// TIA Portal V20 export
FUNCTION_BLOCK "FB_Electrical_Current_Test"   // FB6, LAD
{ S7_Optimized_Access := 'TRUE' }
// stored: MemoryReserve 100, SetENOAutomatically false
   VAR_INPUT
      Star_Functional_Test : Bool;
      Reset_Functional_Test : Bool;
      Electrical_Current_Read_UInt : UInt;
      In_Test_Parameters : "IO_Device_Test_Parameters";
   END_VAR
   VAR_OUTPUT
      Electrical_Current_Test_Approved : Bool;
   END_VAR
   VAR
      Timer_Delay_Read_Current { S7_SetPoint := 'True'} : TON_TIME;
      Timer_Delay_Reset { S7_SetPoint := 'True'} : TON_TIME;
   END_VAR
BEGIN

REGION Network 1
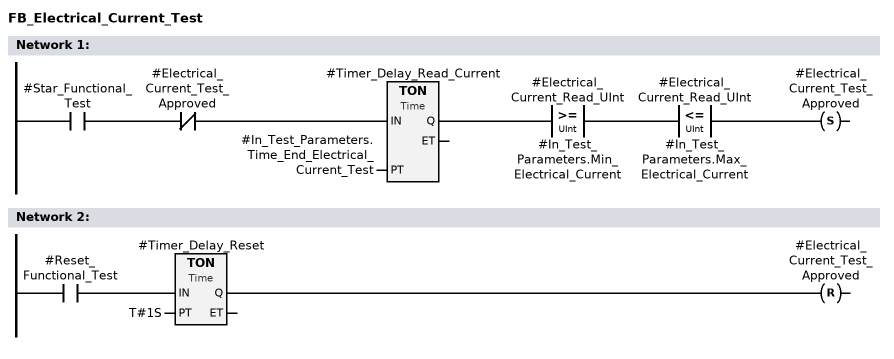
   RUNG wire#powerrail
      Contact( #Star_Functional_Test )
      I_Contact( #Electrical_Current_Test_Approved )
      { S7_Templates := "time_type := Time" } #Timer_Delay_Read_Current.TON(pt := #In_Test_Parameters.Time_End_Electrical_Current_Test, et =>)
      { S7_Templates := "SrcType := UInt" } GE_Contact(in1 := #Electrical_Current_Read_UInt, in2 := #In_Test_Parameters.Min_Electrical_Current)
      { S7_Templates := "SrcType := UInt" } LE_Contact(in1 := #Electrical_Current_Read_UInt, in2 := #In_Test_Parameters.Max_Electrical_Current)
      S_Coil( #Electrical_Current_Test_Approved )
   END_RUNG
   // the same network as SCL:
   #Timer_Delay_Read_Current(IN := #Star_Functional_Test AND NOT #Electrical_Current_Test_Approved,   // TON
                           PT := #In_Test_Parameters.Time_End_Electrical_Current_Test);
   IF #Timer_Delay_Read_Current.Q AND (#Electrical_Current_Read_UInt >= #In_Test_Parameters.Min_Electrical_Current) AND (#Electrical_Current_Read_UInt <= #In_Test_Parameters.Max_Electrical_Current) THEN
       #Electrical_Current_Test_Approved := TRUE;
   END_IF;
END_REGION

REGION Network 2
   RUNG wire#powerrail
      Contact( #Reset_Functional_Test )
      { S7_Templates := "time_type := Time" } #Timer_Delay_Reset.TON(pt := T#1S, et =>)
      R_Coil( #Electrical_Current_Test_Approved )
   END_RUNG
   // the same network as SCL:
   #Timer_Delay_Reset(IN := #Reset_Functional_Test, PT := T#1S);   // TON
   IF #Timer_Delay_Reset.Q THEN #Electrical_Current_Test_Approved := FALSE; END_IF;
END_REGION
END_FUNCTION_BLOCK
